FUNCTION_BLOCK xPlanarPower
VAR_INPUT
	TriggerEnable	: BOOL;
	TriggerDisable	: BOOL;
END_VAR
VAR_OUTPUT
END_VAR
VAR
	Running			: BYTE;
	
	i				: BYTE;
	State			: BYTE;
	CommandDone		: BOOL;
	
	EnableDone		: BOOL;
	DisableDone		: BOOL;
END_VAR


Running := Running + 1;

EnableMovers();

DisableMovers();

ReadPowerStatus();

METHOD DisableMovers : BOOL
VAR_INPUT
END_VAR

IF TriggerDisable THEN
	
	EnableDone := FALSE;

	CASE State OF
		
		0:
			TriggerDisable := FALSE;
			
			FOR i := 1 TO xPlanarLink.MoverCount DO
				xPlanarLink.PlanarMover[i].Disable(xPlanarLink.PlanarFeedback[i]);
			END_FOR
			State := 1;
		
		1:
			FOR i := 1 TO xPlanarLink.MoverCount DO
				CommandDone := xPlanarLink.PlanarFeedback[i].Done;
			END_FOR
			
			IF CommandDone THEN
				CommandDone := FALSE;
				State := 2;
			END_IF
		
		2:
			DisableDone := TRUE;
	
	END_CASE

END_IF
END_METHOD

METHOD EnableMovers : BOOL
VAR_INPUT
END_VAR

IF TriggerEnable THEN

	DisableDone := FALSE;	
	
	CASE State OF
		
		0:
			TriggerEnable := FALSE;
			
			FOR i := 1 TO xPlanarLink.MoverCount DO
				xPlanarLink.PlanarMover[i].Enable(xPlanarLink.PlanarFeedback[i]);
			END_FOR
			State := 1;
		
		1:
			FOR i := 1 TO xPlanarLink.MoverCount DO
				CommandDone := xPlanarLink.PlanarFeedback[i].Done;
			END_FOR
			
			IF CommandDone THEN
				CommandDone := FALSE;
				State := 2;
			END_IF
		
		2:
			EnableDone := TRUE;
	
	END_CASE

END_IF
END_METHOD

METHOD ReadPowerStatus : BOOL
VAR_INPUT
END_VAR

FOR i := 1 TO xPlanarLink.MoverCount DO
	
	IF xPlanarLink.PlanarMover[i].MCTOPLC.STD.State = 3 THEN
		EnableDone := TRUE;
		DisableDone := FALSE;
	ELSE
		DisableDone := TRUE;
		EnableDone := FALSE;
	END_IF

END_FOR
END_METHOD

END_FUNCTION_BLOCK

(* stored: Version 1.1.0.1, ProductVersion 3.1.4024.12
   POU xPlanarPower: Id {c74e6ded-70f6-4dde-a622-675725c54072}, SpecialFunc None
   Method DisableMovers: Id {e7dd4c1b-e93a-42af-bc89-25e44ea8a2fb}
   Method EnableMovers: Id {c0071bb0-05f7-42e7-bc56-2ba89d9785b0}
   Method ReadPowerStatus: Id {7a51f4b8-99c5-4291-a1f9-55d97ad18f46} *)
